Fanuc KAREL source: NC0010.KL

-- PROVISIONAL review KL for V1013-1; original PC SHA256 c1bbeae03c6cf31d24e9d861f5041f791f056c9652b72b6a7980ed00d6a8886c
-- Incomplete behavior may be omitted. Consult companion uncertainty JSON. Do not deploy.
PROGRAM NC0010
%NOLOCKGROUP
-- UNRESOLVED_LOCAL_POOL 1 cells at code offset 3; source declarations unknown
-- DIRECT_LOCAL_WORD_ACCESS alone does not prove INTEGER, REAL, or BOOLEAN
BEGIN
  -- UNRESOLVED_PC offsets 0-8; opcodes 2B,2C,7B
  -- UNRESOLVED_PC offsets 13-20; opcodes 9D,23
  -- UNRESOLVED_PC offsets 25-38; opcodes 21,9D,57,79
  -- UNRESOLVED_PC offsets 43-56; opcodes 21,9D,57,79
  -- UNRESOLVED_PC offsets 61-74; opcodes 21,9D,57,79
  -- UNRESOLVED_PC offsets 79-92; opcodes 21,9D,57,79
  -- UNRESOLVED_PC offsets 97-110; opcodes 21,9D,57,79
  -- UNRESOLVED_PC offsets 115-128; opcodes 21,9D,57,79
  -- UNRESOLVED_PC offsets 133-146; opcodes 21,9D,57,79
  -- UNRESOLVED_PC offsets 151-164; opcodes 21,9D,57,79
  -- UNRESOLVED_PC offsets 169-182; opcodes 21,9D,57,79
  -- UNRESOLVED_PC offsets 187-200; opcodes 21,9D,57,79
  -- UNRESOLVED_PC offsets 205-218; opcodes 21,9D,57,79
  -- UNRESOLVED_PC offsets 223-236; opcodes 21,9D,57,79
  -- UNRESOLVED_PC offsets 241-254; opcodes 21,9D,57,79
  -- UNRESOLVED_PC offsets 259-272; opcodes 21,9D,57,79
  -- UNRESOLVED_PC offsets 277-290; opcodes 21,9D,57,79
  -- UNRESOLVED_PC offsets 295-308; opcodes 21,9D,57,79
  -- UNRESOLVED_PC offsets 313-326; opcodes 21,9D,57,79
  -- UNRESOLVED_PC offsets 331-344; opcodes 21,9D,57,79
  -- UNRESOLVED_PC offsets 349-363; opcodes 21,9D,52,23
  -- UNRESOLVED_PC offsets 368-373; opcodes 7A
  -- UNRESOLVED_PC offsets 378-396; opcodes 21,2E,52,23
  -- UNRESOLVED_PC offsets 406-411; opcodes 7A
  -- UNRESOLVED_PC offsets 416-434; opcodes 21,2E,52,23
  -- UNRESOLVED_PC offsets 444-449; opcodes 7A
  -- UNRESOLVED_PC offsets 454-472; opcodes 21,2E,52,23
  -- UNRESOLVED_PC offsets 482-487; opcodes 7A
  -- UNRESOLVED_PC offsets 492-510; opcodes 21,2E,52,23
  -- UNRESOLVED_PC offsets 520-525; opcodes 7A
  -- UNRESOLVED_PC offsets 530-548; opcodes 21,2E,52,23
  -- UNRESOLVED_PC offsets 558-563; opcodes 7A
  -- UNRESOLVED_PC offsets 568-586; opcodes 21,2E,52,23
  -- UNRESOLVED_PC offsets 596-601; opcodes 7A
  -- UNRESOLVED_PC offsets 606-624; opcodes 21,2E,52,23
  -- UNRESOLVED_PC offsets 634-639; opcodes 7A
  -- UNRESOLVED_PC offsets 644-662; opcodes 21,2E,52,23
  -- UNRESOLVED_PC offsets 672-677; opcodes 7A
  -- UNRESOLVED_PC offsets 682-700; opcodes 21,2E,52,23
  -- UNRESOLVED_PC offsets 710-715; opcodes 7A
  -- UNRESOLVED_PC offsets 720-738; opcodes 21,2E,52,23
  -- UNRESOLVED_PC offsets 748-753; opcodes 7A
  -- UNRESOLVED_PC offsets 758-776; opcodes 21,2E,52,23
  -- UNRESOLVED_PC offsets 786-791; opcodes 7A
  -- UNRESOLVED_PC offsets 796-814; opcodes 21,2E,52,23
  -- UNRESOLVED_PC offsets 824-829; opcodes 7A
  -- UNRESOLVED_PC offsets 834-852; opcodes 21,2E,52,23
  -- UNRESOLVED_PC offsets 862-867; opcodes 7A
  -- UNRESOLVED_PC offsets 872-890; opcodes 21,2E,52,23
  -- UNRESOLVED_PC offsets 900-905; opcodes 7A
  -- UNRESOLVED_PC offsets 910-928; opcodes 21,2E,52,23
  -- UNRESOLVED_PC offsets 938-943; opcodes 7A
  -- UNRESOLVED_PC offsets 948-966; opcodes 21,2E,52,23
  -- UNRESOLVED_PC offsets 976-981; opcodes 7A
  -- UNRESOLVED_PC offsets 986-1004; opcodes 21,2E,52,23
  -- UNRESOLVED_PC offsets 1014-1019; opcodes 7A
  -- UNRESOLVED_PC offsets 1024-1042; opcodes 21,2E,52,23
  -- UNRESOLVED_PC offsets 1052-1056; opcodes 7F
  -- UNRESOLVED_PC offsets 1061-1065; opcodes 27,AA
  -- UNRESOLVED_PC offsets 1070-1074; opcodes 7F
END NC0010
